// Interlock logic for the Baseplate Chiller
FUNCTION F_BaseplateChillerEnable : BOOL
VAR_INPUT
    bMasterOverride : BOOL; //Master manual override control input
END_VAR
VAR_IN_OUT CONSTANT
    stErrors : ST_ErrorStates; // Currently detected errors
END_VAR
VAR
END_VAR

IF (stErrors.bHardwareFailure // Disable baseplate chiller if there is a hardware failure
    OR stErrors.bLeakUnderTable) // Disable baseplate chiller if there is a leak under the table
    AND NOT bMasterOverride //if master override is TRUE, ignore all errors
THEN
    F_BaseplateChillerEnable := FALSE;
ELSE
    F_BaseplateChillerEnable := TRUE;
END_IF

END_FUNCTION

(* stored: Version 1.1.0.1, ProductVersion 3.1.4022.18
   POU F_BaseplateChillerEnable: Id {1364b9de-d1e4-4cd9-be0a-b8eefa4075df}, SpecialFunc None *)
